// TIA Portal V19 export
DATA_BLOCK "Axis_1"   // DB1, Motion_DB
AUTHOR : SIMATIC
FAMILY : BasicMC
NAME : TO_PosAx
VERSION : 7.0
// stored: InstanceOfName TO_PositioningAxis, OfSystemLibElement TO_PositioningAxis, OfSystemLibVersion 7.0
TO_PositioningAxis   // technology object, version 7.0
   // // inherited from TO_SpeedAxis
   // // inherited from TO_Axis
   // // inherited from TO_AnyMotionObject
   // VAR
   //    Header : TO_Struct_Header;
   // END_VAR
   // VAR
   //    Position { ExternalWritable := 'False'} : Real;
   //    Velocity { ExternalWritable := 'False'} : Real;
   //    ActualPosition { ExternalWritable := 'False'} : Real;
   //    ActualVelocity { ExternalWritable := 'False'} : Real;
   //    Actor { S7_SetPoint := 'True'} : TO_Struct_Actor;
   //    Sensor { S7_SetPoint := 'True'} : Array[1..1] of TO_Struct_Sensor;
   //    Units { ExternalWritable := 'False'; S7_SetPoint := 'True'} : TO_Struct_Units;
   //    Mechanics { ExternalWritable := 'False'; S7_SetPoint := 'True'} : TO_Struct_Mechanics;
   //    DynamicLimits { ExternalWritable := 'False'; S7_SetPoint := 'True'} : TO_Struct_DynamicLimits;
   //    DynamicDefaults { S7_SetPoint := 'True'} : TO_Struct_DynamicDefaults;
   //    Modulo { ExternalWritable := 'False'; S7_SetPoint := 'True'} : TO_Struct_Modulo;
   //    PositionLimits_SW { S7_SetPoint := 'True'} : TO_Struct_PositionLimitsSW;
   //    PositionLimits_HW { S7_SetPoint := 'True'} : TO_Struct_PositionLimitsHW;
   //    Homing { S7_SetPoint := 'True'} : TO_Struct_Homing;
   //    PositionControl { ExternalWritable := 'False'; S7_SetPoint := 'True'} : TO_Struct_PositionControl;
   //    FollowingError { ExternalWritable := 'False'; S7_SetPoint := 'True'} : TO_Struct_FollowingError;
   //    PositioningMonitoring { ExternalWritable := 'False'; S7_SetPoint := 'True'} : TO_Struct_PositioningMonitoring;
   //    StandstillSignal { ExternalWritable := 'False'; S7_SetPoint := 'True'} : TO_Struct_StandstillSignal;
   //    Simulation { ExternalWritable := 'False'; S7_SetPoint := 'True'} : TO_Struct_Simulation;
   //    StatusPositioning { ExternalWritable := 'False'; S7_SetPoint := 'True'} : TO_Struct_StatusPositioning;
   //    StatusDrive { ExternalWritable := 'False'; S7_SetPoint := 'True'} : TO_Struct_StatusDrive;
   //    StatusSensor { ExternalWritable := 'False'; S7_SetPoint := 'True'} : Array[1..1] of TO_Struct_StatusSensor;
   //    StatusBits { ExternalWritable := 'False'; S7_SetPoint := 'True'} : TO_Struct_StatusBits;
   //    ErrorBits { ExternalWritable := 'False'; S7_SetPoint := 'True'} : TO_Struct_ErrorBits;
   //    ControlPanel { S7_SetPoint := 'True'} : TO_Struct_ControlPanel;
   //    Internal { S7_SetPoint := 'True'} : Array[1..4] of TO_Struct_Internal;
   // END_VAR
BEGIN
   Header.VersionMaj := 7;
   Header.VersionMin := 0;
   Header."Type" := 1;
   Actor."Type" := 1;
   Actor.DataAdaption := 1;
   Actor.Interface.AddressIn.RID := 16#0208_070C;
   Actor.Interface.AddressIn.AREA := 16#81;
   Actor.Interface.AddressIn.OFFSET := 544;
   Actor.Interface.AddressOut.RID := 16#0208_070D;
   Actor.Interface.AddressOut.AREA := 16#82;
   Actor.Interface.AddressOut.OFFSET := 656;
   Actor.DriveParameter.MaxSpeed := 5000.0;
   Sensor[1].DataAdaption := 1;
   Sensor[1].Interface.AddressIn.RID := 16#0208_070C;
   Sensor[1].Interface.AddressIn.AREA := 16#81;
   Sensor[1].Interface.AddressIn.OFFSET := 544;
   Sensor[1].Interface.AddressOut.RID := 16#0208_070D;
   Sensor[1].Interface.AddressOut.AREA := 16#82;
   Sensor[1].Interface.AddressOut.OFFSET := 656;
   Sensor[1].Interface."Type" := 2;
   Sensor[1].Parameter.StepsPerRevolution := 2500;
   Sensor[1].Parameter.FineResolutionXist1 := 2;
   Sensor[1].Parameter.FineResolutionXist2 := 0;
   Sensor[1].Parameter.DeterminableRevolutions := 0;
   Sensor[1].ActiveHoming.DigitalInputAddress.RID := 16#0200_0001;
   Sensor[1].ActiveHoming.DigitalInputAddress.AREA := 16#81;
   Sensor[1].ActiveHoming.DigitalInputAddress.OFFSET := 3;
   Sensor[1].ActiveHoming.SwitchLevel := FALSE;
   DynamicLimits.MinVelocity := 0.0;
   DynamicDefaults.Acceleration := 50.0;
   DynamicDefaults.Deceleration := 50.0;
   DynamicDefaults.EmergencyDeceleration := 125.0;
   Homing.AutoReversal := FALSE;
   Homing.ApproachDirection := FALSE;
   _Sensor[1].ActiveHoming.DigitalInput := Axis_1_Homing switch;
   _Sensor[1].DataAdaptionOffline := True;
   _Sensor[1].Interface.ProfiDriveOutName := Axis_1_Drive_OUT;
   _Sensor[1].Interface.ProfiDriveInName := Axis_1_Drive_IN;
   _Actor.DataAdaptionOffline := True;
   _Actor.Interface.ProfiDriveOutName := Axis_1_Drive_OUT;
   _Actor.Interface.ProfiDriveInName := Axis_1_Drive_IN;
   _Sensor[1].Interface.EncoderConnection := 7;
END_DATA_BLOCK
